// TIA Portal V19 export
TYPE "PositioningMachine_Manager"
// stored: Access Published
   STRUCT
      EnableStopDoorOpeningReq : Bool := TRUE;
      EnableStopInPhase : Bool := TRUE;
      EnableStopProgrammed : Bool := TRUE;
      Control_ON : Bool := FALSE;
      SelectMotorEncoder : Bool := TRUE;   // TRUE = Use motor encoder (1) / FALSE = Use Measurinf Wheel encoder (2)
      Bwd : Bool := FALSE;
      Fwd : Bool := FALSE;
      MoveToPos : Bool := FALSE;
      UsePositionControl : Bool := FALSE;
      Pos : LReal := 0.0;
      Vel : LReal := 100.0;
      Acc : LReal := 100.0;
      Dec : LReal := 100.0;
      Jerk : LReal := 0.0;
   END_STRUCT;
END_TYPE
